TYPE ST_SettingsDockingClamps :
STRUCT
	tClampsOpenTimeout : TIME := T#10S;	/// Timeout for opening clamps [default: 10s]
	tClampsCloseTimeout : TIME := T#10S;	/// Timeout for closing clamps [default: 10s]
END_STRUCT
END_TYPE

(* stored: Version 1.1.0.1, ProductVersion 3.1.4024.12
   DUT ST_SettingsDockingClamps: Id {3c243beb-1cc1-41a2-bbc8-1c151cff727e} *)
